FUNCTION_BLOCK WELD_ROBOT
VAR_INPUT
	StartPB : BOOL;
	RobotReady : BOOL;
	
	
	RobotFault : BOOL;
	SafetyOK : BOOL;
	WeldProgram : INT;
	ResetPB : BOOL;
	
END_VAR
VAR_OUTPUT
	Eno : BOOL;
	RobotStart : BOOL;
	RobotReset : BOOL;
	RobotBusy : BOOL;
	RobotComplete : BOOL;
	RobotHOME : BOOL;
	ProgBit0 : BOOL;
	ProgBit1 : BOOL;
	ProgBit2 : BOOL;
	ProgBit3 : BOOL;
	
END_VAR
VAR
	ProgNum: INT;
	T_Weld_Time : TON;
	
	AutoRequest : BOOL;
    StartEdge   : R_TRIG;
    CycleRun    : BOOL;
    FaultLamp  : BOOL;
	CycleComplete : BOOL;
	Step : INT;
END_VAR

(*0 = Idle
10 = Send Program Number
20 = Start Robot
30 = Wait Busy
40 = Wait Complete
50 = Cycle Finish
900 = Fault*)
IF NOT SafetyOK THEN Step := 0;
	
END_IF
CASE Step OF

0:   RobotHOME := TRUE;
     //RobotStart := FALSE;
     RobotBusy := FALSE;
	 T_Weld_Time(IN :=FALSE);
	 
	 RobotComplete := FALSE;
    IF StartPB AND SafetyOK THEN
       Step := 10;
    END_IF;

10:
    WeldProgram := 5;
	RobotBusy := TRUE;
	RobotHOME := FALSE;
    Step := 20;

20:
    //RobotStart := TRUE;
	//RobotBusy := FALSE;
	//RobotComplete := TRUE;
	T_Weld_Time(IN := TRUE, PT :=T#5S);
   
    IF T_Weld_Time.Q THEN
       RobotComplete := TRUE; RobotStart := FALSE; RobotBusy := FALSE;
       Step := 30;
    END_IF;

30:
    IF RobotComplete THEN
		//T_Weld_Time.Q :=FALSE;
       Step := 0;
    END_IF;



END_CASE;

END_FUNCTION_BLOCK

(* stored: Version 1.1.0.1, ProductVersion 3.1.4024.16
   POU WELD_ROBOT: Id {2349e916-c386-4bf9-be6b-d9f1c8805cd4}, SpecialFunc None *)
